# B&R Automation Studio project SuperTrak_Core (part 2)

#### actWidgets.st
```iecst
ACTION SuperTrakPaperWidget:

	WidgetData.SectionCount	:= CONFIG_ST_MAX_SECTIONS;
	WidgetData.ShuttleCount := gSuperTrak.Status.System.ActivePallets;

	FOR index := 1 TO gSuperTrak.Status.System.ActivePallets DO
		// Calculate pallet position in terms of total distance along track- including some scaling for Curve Sections
		IF gSuperTrak.Status.Section[gSuperTrak.Status.Pallet[index].Section].IsCurveSection = FALSE THEN
			WidgetData.ShuttlePos[index]			:= 	(UINT_TO_REAL(gSuperTrak.Status.Pallet[index].Section) - 1.0) * (1000.0) +
			(gSuperTrak.Status.Pallet[index].Position / 1000.0) * (1000.0);
		ELSE
			WidgetData.ShuttlePos[index]			:= 	(UINT_TO_REAL(gSuperTrak.Status.Pallet[index].Section) - 1.0) * (1000.0) +
			(gSuperTrak.Status.Pallet[index].Position / 1030.0) * (1000.0);
		END_IF;
	END_FOR;

	WidgetData.TargetCount	:= 0;

	FOR index := 1 TO CONFIG_ST_MAX_TARGETS DO

		IF gSuperTrak.Status.Target[index].Section <> 0 THEN
			WidgetData.TargetCount		:= WidgetData.TargetCount + 1;
		END_IF;

		// Calculate target position in terms of total distance along track- including some scaling for Curve Sections
		IF gSuperTrak.Status.Section[gSuperTrak.Status.Target[index].Section].IsCurveSection = FALSE THEN
			WidgetData.TargetPos[index]				:= (UINT_TO_REAL(gSuperTrak.Status.Target[index].Section) - 1.0) * (1000.0) +
			(gSuperTrak.Status.Target[index].Position / 1000.0) * (1000.0);
		ELSE
			WidgetData.TargetPos[index]				:= (UINT_TO_REAL(gSuperTrak.Status.Target[index].Section) - 1.0) * (1000.0) +
			(gSuperTrak.Status.Target[index].Position / 1030.0) * (1000.0);
		END_IF;
	END_FOR;

	pTargetStatusRef		ACCESS ADR(gSuperTrak.Status.Target[targetStatusIndex+1]);
	pSectionStatusRef		ACCESS ADR(gSuperTrak.Status.Section[sectionStatusIndex+1]);
	pPalletStatusRef		ACCESS ADR(gSuperTrak.Status.Pallet[palletStatusIndex+1]);

END_ACTION
```

### Program Logical/Source/ST_Core/ST_Main_OLD

#### Variables.var
```iecst
(********************************************************************
 * Copyright ATS Automation Tooling Systems, Inc. 2015
 * All rights reserved.
 ********************************************************************
 * Local variables
 ********************************************************************)
VAR
	i : USINT := 0;
	ServiceChannelData : ServiceChannel_t := (0);
	pResView : REFERENCE TO ServiceChannelHeader_t;
	pReqView : REFERENCE TO ServiceChannelHeader_t;
	SuperTrakControlInterface : ARRAY[0..stMAX_CONTROL_IF_INDEX] OF SuperTrakControlInterface_t := [stMAX_CONTROL_IF_COUNT((0))];
	DeviceDetectInterface0 : DeviceDetectInterface := (0);
	mvCounter : INT;
	IsSimulation : BOOL;
	taskName : STRING[80];
	status : UINT;
	taskGroup : USINT;
	SuperTrakStoragePath : STRING[80];
END_VAR
```

#### Main.st
```iecst
(*********************************************************************************
 * Copyright: ATS Automation Tooling Systems, Inc. 2015
 *     All rights reserved.
 *********************************************************************************
 *********************************************************************************
 * Description:
 * -------------------------------------------------------------------------------
 * This task configures the internal communication structure AND controlls
 * the SuperTrak system.
 *********************************************************************************)

PROGRAM _INIT

	testString;

	(* DiagCpuIsSimulated() returns TRUE if "Activate Simulation" is enabled. *)
	IsSimulation := DiagCpuIsSimulated();

	(* DiagCpuIsSimulated() returns FALSE if the project configuration specifies
	 * ARsim. Assume simulation mode IF this task is named 'ST_MainSim'.
	 *)
	taskName := '';
	status := ST_name(0, ADR(taskName), ADR(taskGroup));

	IF (taskName = 'ST_MainSim') THEN
		IsSimulation := TRUE;
	END_IF;

	IF (IsSimulation) THEN
		(* This path can be customized as needed *)
		SuperTrakStoragePath := '/DEVICE=../../../../Logical/ConfigFiles';
		//SuperTrakStoragePath	:= '/DEVICE=C:\SuperTrakCfg\SuperTrakCore';
	ELSE
		(* CFast card USER partition *)
		SuperTrakStoragePath := '/DEVICE=F:\SuperTrakCore';
	END_IF;

	// SuperTrak initialization
	SuperTrakInit(IsSimulation,SuperTrakStoragePath);

	DeviceDetectInterface0.allowConfiguration  := TRUE;
	DeviceDetectInterface0.deviceState    := 1;
	DeviceDetectInterface0.deviceType    := DEVICE_TYPE_SUPERTRAK_G3;
	DeviceDetectInterface0.enable     := TRUE;
	DeviceDetectInterface0.device     := ''; (* empty for ARsim *)
	DeviceDetectInterface0();

	// Service Channel initialization
	ServiceChannelData.channelId    		:= 1;
	ServiceChannelData.pRequestHeader		:= ADR(gStServiceChannelReqData);
	ServiceChannelData.pResponseHeader		:= ADR(gStServiceChannelResData);
	ServiceChannelData.pRequestValues     	:= ADR(gStServiceChannelReqData) + SIZEOF(ServiceChannelHeader_t);
	ServiceChannelData.pResponseValues    	:= ADR(gStServiceChannelResData) + SIZEOF(ServiceChannelHeader_t);
	ServiceChannelData.requestBufferSize  	:= SIZEOF(gStServiceChannelReqData);
	ServiceChannelData.responseBufferSize  	:= SIZEOF(gStServiceChannelResData);
	ServiceChannelData.state     			:= scSTATE_RECV;

	pResView ACCESS ADR(gStServiceChannelResData);
	pReqView ACCESS ADR(gStServiceChannelReqData);

	// Command interface mapping
	SuperTrakControlInterface[0].pControl   := ADR(gStCyclicControlData);
	SuperTrakControlInterface[0].pStatus   := ADR(gStCyclicStatusData);
	SuperTrakControlInterface[0].controlSize  := SIZEOF(gStCyclicControlData);
	SuperTrakControlInterface[0].statusSize  := SIZEOF(gStCyclicStatusData);

	mvCounter;

END_PROGRAM

PROGRAM _CYCLIC

	mvCounter := mvCounter + 1;

	// Cyclic SuperTrak control
	SuperTrakCyclic();

	// Map internal communication structure
	FOR i := 0 TO stMAX_CONTROL_IF_INDEX DO
		SuperTrakProcessControl(i, SuperTrakControlInterface[i]);
	END_FOR;

	// Service channel handling
	IF ServiceChannelData.state = scSTATE_RECV AND
		pReqView.sequence <> pResView.sequence THEN
		ServiceChannelData.requestSequence  := pReqView.sequence;
		ServiceChannelData.state    		:= scSTATE_EXEC;
	ELSIF ServiceChannelData.state = scSTATE_EXEC OR ServiceChannelData.state = scSTATE_WAIT THEN
		SuperTrakServiceChannel(ServiceChannelData);
	ELSIF ServiceChannelData.state = scSTATE_SEND THEN
		ServiceChannelData.state    		:= scSTATE_RECV;
	END_IF;

END_PROGRAM

PROGRAM _EXIT

 // Clear internal memory
	SuperTrakExit();

END_PROGRAM
```

### Package Logical/Source/Main - Main Application Functionality

### Program Logical/Source/Main/MainCtrl (IEC) - Main state machine

#### Types.typ
```iecst
TYPE
	MainState_enum :
		( (*State machine for main application*)
		DISABLED, (*SuperTrak is powered Off*)
		BEGIN_ENABLE, (*SuperTrak is powering On*)
		START_RECOVERY, (*Begin pallet recovery operation*)
		PALLETS_RECOVERING, (*Pallets currently moving to a recovery target*)
		BEGIN_STOP, (*Single-cycle state to set controlled-stop behavior*)
		STOPPING, (*System executing a controlled stop*)
		READY, (*Powering complete. Ready to begin pallet routing*)
		RUN, (*Pallet routing active*)
		ERROR, (*System in error mode*)
		RESETTING, (*System resetting from error condition*)
		TEST (*Empty case in state machine for debugging through watch window*)
		);
END_TYPE
```

#### Variables.var
```iecst
VAR
	MainState : MainState_enum;
	index : UINT;
	targetTimer : ARRAY[0..20] OF TON;
	systemAccel : UINT := 0;
	systemVelo : UINT := 0;
	nextTarget : USINT;
	blueZoneClear : BOOL;
END_VAR
```

#### Main.st
```iecst
PROGRAM _INIT

	// Recovery positions can be utilized by start logic. By default, these values are utilized by the Pallets Recovering state.
	gSuperTrak.Par.System.RecoveryAccel			:= 2000;
	gSuperTrak.Par.System.RecoveryVelocity		:= 500;
	gSuperTrak.Par.System.RecoveryDirection		:= stCOM_DIR_RIGHT;
	gSuperTrak.Par.System.RecoveryTarget		:= 2;

	systemAccel		:= 20000;
	systemVelo		:= 2000;

	FOR index := 1 TO 20 DO
		targetTimer[index].PT				:= t#500ms;
	END_FOR;

	nextTarget	:= 5;

END_PROGRAM

PROGRAM _CYCLIC

	// Return the state machine to a DISABLED state when the system stops itself
	gSuperTrak.Status.System.Running				:= FALSE;
	IF gSuperTrak.Status.System.Enabled = FALSE THEN
		MainState									:= DISABLED;
	END_IF;

	// Return the state machine to a DISABLED state when commanded
	IF gSuperTrak.Cmds.Enable = FALSE THEN
		MainState									:= DISABLED;
	END_IF;

	// Primary state machine for the SuperTrak
	CASE MainState OF
		DISABLED://======================================================================================
			// System is unpowered. Track sections disabled
			// If stuck in this state, check that ST_CONFIG_MAX_SECTIONS is configured correctly

			gSuperTrak.Cmds.Start					:= FALSE;
			IF gSuperTrak.Cmds.Enable THEN
				MainState							:= BEGIN_ENABLE;
			END_IF;

		BEGIN_ENABLE://======================================================================================
			// Confirm system response

			IF gSuperTrak.Status.System.Enabled THEN
				MainState							:= START_RECOVERY;
			END_IF;

		START_RECOVERY://====================================================================================
			// Application-specific recovery logic can be built here. Based on default logic, shuttles need to reach their commanded
			// target to be considered 'ready'. Pallets in queue are not considered fully recovered.

			MainState								:= PALLETS_RECOVERING;

		PALLETS_RECOVERING://======================================================================================
			// Confirm system response. Move shuttles away from the Load Target so that trailing shuttles can reach this position also

			IF gSuperTrak.Status.Target[1].PalletPresent THEN

				gSuperTrak.Par.Target[1].Config.Acceleration		:= gSuperTrak.Par.System.RecoveryAccel;
				gSuperTrak.Par.Target[1].Config.Velocity			:= gSuperTrak.Par.System.RecoveryVelocity;
				gSuperTrak.Par.Target[1].Config.DestinationTarget	:= gSuperTrak.Par.System.RecoveryTarget;
				gSuperTrak.Par.Target[1].Config.Direction			:= gSuperTrak.Par.System.RecoveryDirection;

				gSuperTrak.Par.Target[1].ReleaseToTarget		:= TRUE;
			ELSE
				gSuperTrak.Par.Target[1].ReleaseToTarget			:= FALSE;
			END_IF;

			// All sections must clear the 'Pallets Recovering' state to enter a Ready mode
			IF gSuperTrak.Status.System.Ready THEN
				MainState							:= READY;
			END_IF;

		READY://======================================================================================
			// System ready. Pallets located. Await RUN command.

			IF gSuperTrak.Cmds.Start THEN
				MainState							:= RUN;
				gSuperTrak.Status.System.Running	:= TRUE;
			END_IF;

		RUN://======================================================================================
			// RUN state. Application pallet routing goes here.

			gSuperTrak.Status.System.Running		:= TRUE;
			IF gSuperTrak.Cmds.Start = FALSE THEN
				MainState							:= BEGIN_STOP;
			END_IF;

			FOR index := 1 TO 20 DO
				targetTimer[index].IN				:= FALSE;
			END_FOR;

			//	----------------------------------------------------------------------- target 1

			IF gSuperTrak.Status.Target[1].PalletPresent THEN

				targetTimer[1].IN		:= TRUE;

				IF targetTimer[1].Q THEN
					gSuperTrak.Par.Target[1].Config.Acceleration		:= systemAccel;
					gSuperTrak.Par.Target[1].Config.Velocity			:= systemVelo;
					gSuperTrak.Par.Target[1].Config.DestinationTarget	:= 2;
					gSuperTrak.Par.Target[1].Config.Direction			:= stCOM_DIR_RIGHT;

					gSuperTrak.Par.Target[1].ReleaseToTarget			:= TRUE;
				END_IF;
			ELSE
				gSuperTrak.Par.Target[1].ReleaseToTarget				:= FALSE;
			END_IF;

			//	----------------------------------------------------------------------- target 2

			IF gSuperTrak.Status.Target[2].PalletPresent THEN
				targetTimer[2].IN			:= TRUE;

				IF targetTimer[2].Q THEN
					gSuperTrak.Par.Target[2].Config.Acceleration		:= systemAccel;
					gSuperTrak.Par.Target[2].Config.Velocity			:= systemVelo;
					gSuperTrak.Par.Target[2].Config.DestinationTarget	:= 3;
					gSuperTrak.Par.Target[2].Config.Direction			:= stCOM_DIR_RIGHT;

					gSuperTrak.Par.Target[2].ReleaseToTarget		:= TRUE;
				END_IF;

			ELSE
				gSuperTrak.Par.Target[2].ReleaseToTarget			:= FALSE;
			END_IF;

			//	----------------------------------------------------------------------- target 3

			IF EDGENEG( gSuperTrak.Status.Target[3].PalletPresent ) THEN
				CASE nextTarget OF
					4:	nextTarget := 5;
					5:	nextTarget := 4;
				END_CASE;
			END_IF;

			IF gSuperTrak.Status.Target[3].PalletPresent THEN
				targetTimer[3].IN			:= TRUE;

				IF targetTimer[3].Q THEN
					gSuperTrak.Par.Target[3].Config.Acceleration		:= systemAccel;
					gSuperTrak.Par.Target[3].Config.Velocity			:= systemVelo;
					gSuperTrak.Par.Target[3].Config.DestinationTarget	:= nextTarget;
					gSuperTrak.Par.Target[3].Config.Direction			:= stCOM_DIR_RIGHT;

					gSuperTrak.Par.Target[3].ReleaseToTarget		:= TRUE;
				END_IF;

			ELSE
				gSuperTrak.Par.Target[3].ReleaseToTarget			:= FALSE;
			END_IF;

			//	----------------------------------------------------------------------- targets 4 & 5

			IF gSuperTrak.Status.Target[4].PalletPresent AND gSuperTrak.Status.Target[5].PalletPresent THEN

				targetTimer[4].IN			:= TRUE;

				IF targetTimer[4].Q THEN
					gSuperTrak.Par.Target[5].Config.Acceleration		:= systemAccel;
					gSuperTrak.Par.Target[5].Config.Velocity			:= systemVelo;
					gSuperTrak.Par.Target[5].Config.DestinationTarget	:= 6;
					gSuperTrak.Par.Target[5].Config.Direction			:= stCOM_DIR_RIGHT;

					gSuperTrak.Par.Target[4].Config.Acceleration		:= systemAccel;
					gSuperTrak.Par.Target[4].Config.Velocity			:= systemVelo;
					gSuperTrak.Par.Target[4].Config.DestinationTarget	:= 6;
					gSuperTrak.Par.Target[4].Config.Direction			:= stCOM_DIR_RIGHT;

					gSuperTrak.Par.Target[4].ReleaseToTarget		:= TRUE;
					gSuperTrak.Par.Target[5].ReleaseToTarget		:= TRUE;
				END_IF;
			ELSE
				gSuperTrak.Par.Target[4].ReleaseToTarget		:= FALSE;
				gSuperTrak.Par.Target[5].ReleaseToTarget		:= FALSE;
			END_IF;

			//	----------------------------------------------------------------------- target 6

			blueZoneClear		:= TRUE;
			FOR index := 0 TO CONFIG_ST_MAX_PALLETS DO
				IF gSuperTrak.Status.Pallet[index].Section = 2 THEN
					blueZoneClear	:= FALSE;
				END_IF;
			END_FOR;

			IF gSuperTrak.Status.Target[6].PalletPresent AND blueZoneClear THEN
				targetTimer[6].IN			:= TRUE;

				IF targetTimer[6].Q THEN
					gSuperTrak.Par.Target[6].Config.Acceleration		:= systemAccel;
					gSuperTrak.Par.Target[6].Config.Velocity			:= systemVelo;
					gSuperTrak.Par.Target[6].Config.DestinationTarget	:= 2;
					gSuperTrak.Par.Target[6].Config.Direction			:= stCOM_DIR_RIGHT;

					gSuperTrak.Par.Target[6].ReleaseToTarget		:= TRUE;
				END_IF;

			ELSE
				gSuperTrak.Par.Target[6].ReleaseToTarget			:= FALSE;
			END_IF;

			gSuperTrak.Status.Target[1].PalletId;

			(****************	ENTER TARGET LOGIC HERE		****************)

			//			IF gSuperTrak.Status.Target[targetNum].PalletPresent THEN
			//				targetTimer[targetNum].IN			:= TRUE;
			//
			//				IF targetTimer[targetNum].Q THEN
			//					gSuperTrak.Par.Target[targetNum].Config.Acceleration		:= systemAccel;
			//					gSuperTrak.Par.Target[targetNum].Config.Velocity			:= systemVelo;
			//					gSuperTrak.Par.Target[targetNum].Config.DestinationTarget	:= destination;
			//					gSuperTrak.Par.Target[targetNum].Config.Direction			:= stCOM_DIR_RIGHT;
			//
			//					gSuperTrak.Par.Target[targetNum].ReleaseToTarget		:= TRUE;
			//				END_IF;
			//
			//			ELSE
			//				gSuperTrak.Par.Target[targetNum].ReleaseToTarget			:= FALSE;
			//			END_IF;

			//----------------------------------------------------------------

		BEGIN_STOP://==========================================================================================
			// Single-tick state for setting system stop commands

			FOR index := 1 TO CONFIG_ST_MAX_PALLETS DO
				gSuperTrak.Par.Target[index].ReleaseToTarget						:= FALSE;
			END_FOR;

			FOR index := 1 TO CONFIG_ST_MAX_PALLETS DO
				IF gSuperTrak.Status.Pallet[index].PalletAllocated THEN

					gSuperTrak.Par.Pallet[index].Config.Acceleration				:= gSuperTrak.Par.System.RecoveryAccel;
					gSuperTrak.Par.Pallet[index].Config.Velocity					:= gSuperTrak.Par.System.RecoveryVelocity;
					gSuperTrak.Par.Pallet[index].Config.DestinationTarget			:= gSuperTrak.Par.System.RecoveryTarget;
					gSuperTrak.Par.Pallet[index].Config.Direction					:= gSuperTrak.Par.System.RecoveryDirection;

					gSuperTrak.Par.Pallet[index].ReleaseToTarget					:= TRUE;

				END_IF;
			END_FOR;

			MainState															:= STOPPING;

		STOPPING://========================================================================================
			// Application halt logic goes here.

			FOR index := 0 TO CONFIG_ST_MAX_PALLETS DO
				gSuperTrak.Par.Pallet[index].ReleaseToTarget						:= FALSE;
			END_FOR;

			MainState																:= READY;

		ERROR://==========================================================================================
			// Empty state. Placeholder for additional application logic.

		RESETTING://======================================================================================
			// Empty state. Placeholder for additional application logic.

		TEST://===========================================================================================
		// Empty state. Enter for debugging purposes.

	END_CASE;

	// Function block calls
	FOR index := 0 TO 20 DO
		targetTimer[index]();
	END_FOR;

END_PROGRAM
```

### Program Logical/Source/Main/Alarms (IEC) - Handles alarms along with MpAlarmX

#### Main.st - Init, cyclic, exit code
```iecst
PROGRAM _INIT
	(* Insert code here *)

END_PROGRAM

PROGRAM _CYCLIC

	MpAlarmXCore_0(MpLink := ADR(gAlarmXCore), Enable :=TRUE , ErrorReset := gSuperTrak.Cmds.ErrorReset );
	MpAlarmXHistory_0(MpLink :=ADR(gAlarmXHistory) , Enable :=TRUE , ErrorReset :=gSuperTrak.Cmds.ErrorReset , DeviceName := ADR('alarmHistory'), Language := ADR('en'));
	MpAlarmXHistoryUI_0(MpLink :=ADR(gAlarmXHistory) , Enable :=TRUE , ErrorReset :=gSuperTrak.Cmds.ErrorReset, UIConnect := ADR(MpAlarmHistoryUIConnect));
	MpAlarmXListUI_0(MpLink :=ADR(gAlarmXCore) , Enable :=TRUE , ErrorReset :=gSuperTrak.Cmds.ErrorReset, UIConnect :=ADR(MpAlarmUIConnect) );

	// ======================== FAULTS =============================

	FOR index := 0 TO 31 DO

		// Clear value of Reporting Sections string
		nxt_adr		:= memset(ADR(reportingSections),0,SIZEOF(reportingSections)-1);

		IF gSuperTrak.Status.System.Faults[index] THEN
			reportingSections		:= 'System; ';
		END_IF;

		FOR index2 := 0 TO CONFIG_ST_MAX_SECTIONS DO
			IF gSuperTrak.Status.Section[index2].Diag.Faults[index] THEN

				sectionString		:= 'Section ';
				appendString		:= USINT_TO_STRING(index2);

				nxt_adr				:= strcat(ADR(sectionString),ADR(appendString));
				nxt_adr				:= strcat(ADR(sectionString),ADR('; '));
				nxt_adr				:= strcat(ADR(reportingSections),ADR(sectionString));

			END_IF;
		END_FOR;

		alarmString					:= 'Fault_';
		indexString					:= USINT_TO_STRING(index);
		nxt_adr						:= strcat(ADR(alarmString),ADR(indexString));

		IF reportingSections <> '' THEN
			MpAlarmXSet(gAlarmXCore,alarmString);
		ELSE
			MpAlarmXReset(gAlarmXCore,alarmString);
		END_IF;

		IF gSuperTrak.Cmds.ErrorReset THEN
			MpAlarmXAcknowledge(gAlarmXCore,alarmString);
		END_IF;

	END_FOR;

	// ===================== WARNINGS ===========================

	FOR index := 0 TO 31 DO

		// Clear value of Reporting Sections String
		nxt_adr				:= memset(ADR(reportingSections),0,SIZEOF(reportingSections)-1);

		IF gSuperTrak.Status.System.Warnings[index] THEN
			reportingSections			:= 'System; ';
		END_IF;

		FOR index2 := 0 TO CONFIG_ST_MAX_SECTIONS DO
			IF gSuperTrak.Status.Section[index2].Diag.Warnings[index] THEN

				sectionString			:= 'Section ';
				appendString			:= USINT_TO_STRING(index2);

				nxt_adr					:= strcat(ADR(sectionString),ADR(appendString));
				nxt_adr					:= strcat(ADR(sectionString),ADR('; '));
				nxt_adr					:= strcat(ADR(reportingSections),ADR(sectionString));

			END_IF;
		END_FOR;

		alarmString						:= 'Warning_';
		indexString						:= USINT_TO_STRING(index);
		nxt_adr							:= strcat(ADR(alarmString),ADR(indexString));

		IF reportingSections <> '' THEN
			MpAlarmXSet(gAlarmXCore,alarmString);
		ELSE
			MpAlarmXReset(gAlarmXCore,alarmString);
		END_IF;

		IF gSuperTrak.Cmds.ErrorReset THEN
			MpAlarmXAcknowledge(gAlarmXCore,alarmString);
		END_IF;

	END_FOR;

	//========================================================================================================

	(*use this for setting a value through a button on the screen and you want the value that was set to be reset*)
	IF (MpAlarmXHistory_0.Export AND MpAlarmXHistory_0.CommandDone) THEN
		MpAlarmXHistory_0.Export :=	FALSE;
	END_IF

	END_PROGRAM
```

#### Variables.var - Local variables
```iecst
VAR
	MpAlarmXCore_0 : MpAlarmXCore;
	MpAlarmXHistory_0 : MpAlarmXHistory;
	MpAlarmXHistoryUI_0 : MpAlarmXHistoryUI;
	MpAlarmXListUI_0 : MpAlarmXListUI;
	MpAlarmHistoryUIConnect : MpAlarmXHistoryUIConnectType;
	MpAlarmUIConnect : MpAlarmXListUIConnectType;
	index : USINT;
	alarmString : STRING[100];
	nxt_adr : UDINT;
	indexString : STRING[100];
	reportingSections : STRING[100];
	index2 : USINT;
	sectionString : STRING[80];
END_VAR
VAR RETAIN
	appendString : STRING[80];
END_VAR
```

- Visualisation Logical/mappView (not shown)


### Package Logical/ExternalTools - Additional Tools

- MappView.lnk - Links to the mappView page in Chrome (binary file, 2828 bytes)
- AS4_HW_5ACPCE.FMIO-K01.exe (binary file, 355892 bytes)
- ST_6001.dat (binary file, 464508 bytes)
- ST_2000.dat (binary file, 1485820 bytes)
Listed in the project but not available here: Logical/Source/Main/Alarms/Types.typ
